{attribute 'GeneratedUsingTerminal: EL6201-0000-0017'}
{attribute addProperty BoxType "EL6201-0000-0017"}
{attribute addProperty Id "Slave_4A_DO0BOOL1Slave_4A_DO1BOOL1Slave_4A_DO2BOOL1Slave_4A_DO3BOOL1Slave_4B_DO0BOOL1Slave_4B_DO1BOOL1Slave_4B_DO2BOOL1Slave_4B_DO3BOOL1"}
{attribute addProperty CRC "890967761"}
{attribute addProperty Size "8"}
TYPE Slave_4_Outputs_351B16D1 :
STRUCT
	{attribute addProperty Name "Slave_4A_DO0"}
	Slave_4A_DO0 : BOOL;
	{attribute addProperty Name "Slave_4A_DO1"}
	Slave_4A_DO1 : BOOL;
	{attribute addProperty Name "Slave_4A_DO2"}
	Slave_4A_DO2 : BOOL;
	{attribute addProperty Name "Slave_4A_DO3"}
	Slave_4A_DO3 : BOOL;
	{attribute addProperty Name "Slave_4B_DO0"}
	Slave_4B_DO0 : BOOL;
	{attribute addProperty Name "Slave_4B_DO1"}
	Slave_4B_DO1 : BOOL;
	{attribute addProperty Name "Slave_4B_DO2"}
	Slave_4B_DO2 : BOOL;
	{attribute addProperty Name "Slave_4B_DO3"}
	Slave_4B_DO3 : BOOL;
END_STRUCT
END_TYPE

(* stored: Version 1.2.0.0, ProductVersion 3.1.4024.9
   DUT Slave_4_Outputs_351B16D1: Id {599b70a1-d3b2-4430-b098-6d78f20e7bc9} *)
